PROGRAM MAIN
VAR
END_VAR

prgFileWrite();
prgFileRead();

END_PROGRAM

(* stored: Version 1.1.0.1, ProductVersion 3.1.4024.13
   POU MAIN: Id {a95ad861-0ecb-4a03-92c5-4fa259c6e2c9}, SpecialFunc None *)
